{attribute addProperty BoxType "EL5151-0000-0016"}
{attribute addProperty Id "StatusAT %I*Status_690D007D1621Counter_valueAT %I*UDINT32417Latch_valueAT %I*UDINT32418"}
{attribute addProperty CRC "761079895"}
{attribute addProperty SizeInBites "80"}
{attribute addProperty SizeInBytes "10"}
TYPE ENC_Inputs_2D5D2857 :
STRUCT
	{attribute addProperty Name "Status"}
	Status AT %I* : Status_690D007D;
	{attribute addProperty Name "Counter_value"}
	Counter_value AT %I* : UDINT;
	{attribute addProperty Name "Latch_value"}
	Latch_value AT %I* : UDINT;
END_STRUCT
END_TYPE

(* stored: Version 1.2.0.0, ProductVersion 3.1.4024.9
   DUT ENC_Inputs_2D5D2857: Id {049918a3-66d8-4a6b-8679-2a660a7ea39d} *)
